(* PLC project Unnamed, Unknown Unnamed 1 *)
(* stored: creationDateTime 2021-09-19T15:56:13, modificationDateTime 2021-09-19T16:13:59 *)

PROGRAM program0
  VAR
    TON0 : TON;
    LocalVar1 : BOOL;
    LocalVar2 : BOOL;
    Timer : TIME;
    Timer0 : TIME;
  END_VAR

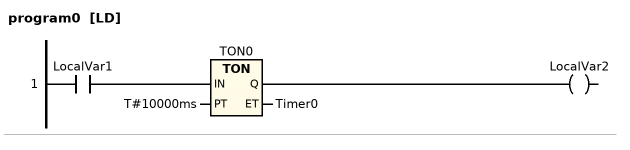
(* LD diagram, written out as Structured Text *)
TON0(IN := LocalVar1, PT := T#10000ms);
LocalVar2 := TON0.Q;
Timer0 := TON0.ET;
END_PROGRAM

CONFIGURATION Config0
  RESOURCE Res0 ON PLC
    TASK task0(INTERVAL := T#20ms, PRIORITY := 0);
    PROGRAM instance0 WITH task0 : program0;
  END_RESOURCE
END_CONFIGURATION
